FUNCTION_BLOCK FB_SimActuator
VAR_INPUT
END_VAR
VAR_OUTPUT
END_VAR
VAR
	bExtended			AT %Q* : BOOL;
	bRetracted			AT %Q* : BOOL := TRUE;
	bExtendCmd			AT %I* : BOOL;
	bRetractCmd			AT %I* : BOOL;
	
	State				: DINT;
	tmrExtend			: TON;
	tmrRetract			: TON;
	iExtendMs			: DINT;
	iRetractMs			: DINT;
	rand				: DRAND;
END_VAR

rand(Seed:=TO_INT(iExtendMs + iRetractMs));
CASE State OF
	0:
		IF bExtendCmd THEN
			iExtendMs := TO_DINT(1500 + (rand.Num * 500));
			State := 1;
		END_IF
		
		IF bRetractCmd THEN
			iRetractMs := TO_DINT(1500 + (rand.Num * 500));
			State := 2;
		END_IF
		
	1:
		tmrExtend(IN:=TRUE, PT:=TO_TIME(iExtendMs));
		IF TO_DINT(tmrExtend.PT) > rand.Num * 100 THEN
			bRetracted := FALSE;
		END_IF
		IF tmrExtend.Q THEN
			bExtended := TRUE;
			tmrExtend(IN:=FALSE);
			State := 0;
		END_IF
		
	2:
		tmrRetract(IN:=TRUE, PT:=TO_TIME(iRetractMs));
		IF TO_DINT(tmrRetract.PT) > rand.Num * 100 THEN
			bExtended := FALSE;
		END_IF
		IF tmrRetract.Q THEN
			bRetracted := TRUE;
			tmrRetract(IN:=FALSE);
			State := 0;
		END_IF
		
END_CASE

END_FUNCTION_BLOCK

(* stored: Version 1.1.0.1, ProductVersion 3.1.4024.12
   POU FB_SimActuator: Id {241a69ff-e48a-46bd-998c-79482a295d18}, SpecialFunc None *)
